FUNCTION_BLOCK LevelSetPoint (* Basic Function Block Type *)
  (* Standard: 61499-2 *)
  (* Version 0.0, 6/10/2026, Schneider Electric, Template *)
  PACKAGE SE.Nereda;
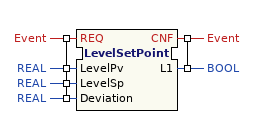
  EVENT_INPUT
    REQ WITH LevelSp, LevelPv, Deviation; (* Normal Execution Request *)
  END_EVENT
  EVENT_OUTPUT
    CNF WITH L1; (* Execution Confirmation *)
  END_EVENT
  VAR_INPUT
    LevelPv : REAL; (* Input event qualifier *)
    LevelSp : REAL;
    Deviation : REAL;
  END_VAR
  VAR_OUTPUT
    L1 : BOOL; (* Output event qualifier *)
  END_VAR
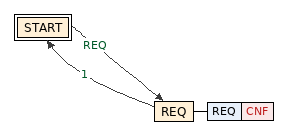
  EC_STATES
    START; (* Initial State *)
    REQ : REQ -> CNF; (* Normal execution *)
  END_STATES
  EC_TRANSITIONS
    START TO REQ := REQ;
    REQ TO START := 1;
  END_TRANSITIONS
  ALGORITHM REQ IN ST: (* Normally executed algorithm *)
;
IF (LevelPv <= LevelSp - Deviation) THEN
	L1 := TRUE;
ELSE
	L1 := FALSE;
END_IF;
  END_ALGORITHM
END_FUNCTION_BLOCK
